{attribute 'estimated-stack-usage' := '4096'}
FUNCTION F_ReadRawMessage : HRESULT
VAR_IN_OUT
    fbCtx   : FB_ParseContext;     
END_VAR
VAR_INPUT
    iMessage : I_Message;
END_VAR
VAR
    iBufferMessage : I_BufferMessage;
    refState : REFERENCE TO ST_ParserInternalState;
END_VAR


refState REF= fbCtx.refCtx.stState;

IF iMessage = 0 THEN
    F_ReadRawMessage := refState.eParserErrorCode := E_ParserErrorCode.InternalError;
    refState.bError := TRUE;
    RETURN;
END_IF

IF __QUERYINTERFACE(iMessage, iBufferMessage) THEN

    F_ReadRawMessage := iBufferMessage.InternalMergeFrom(fbCtx);
    RETURN;
  
ELSE
    IF refState.pCodedInputStream = NULL THEN
        F_ReadRawMessage := refState.eParserErrorCode := E_ParserErrorCode.InternalError;
        refState.bError := TRUE;
        RETURN;
    END_IF
    fbCtx.CopyStateToInputStream(fbInputStream:= refState.pCodedInputStream^);
    iMessage.MergeFrom(fbInput:= refState.pCodedInputStream^);
    fbCtx.LoadStateFromInputStream(fbInputStream:= refState.pCodedInputStream^);
END_IF

END_FUNCTION

(* stored: Version 1.1.0.1
   POU F_ReadRawMessage: Id {c47d844f-4687-416d-9a60-b87fd3566db4}, SpecialFunc None *)
